// TIA Portal V18 export
DATA_BLOCK "Var_HMI"   // DB10
{ S7_Optimized_Access := 'FALSE' }
VERSION : 0.1
// stored: AutoNumber true, IsOnlyStoredInLoadMemory false, IsWriteProtectedInAS false
   VAR
      "popup Emergency" : Bool;
      "popup warning" : Bool;
      Selector : UInt := 5;
      "page number" : UInt := 12;
      in_selection : Bool;
      emergency_popup : Bool;
      selection_no : Int;
      scrolling_1 : Int;
      scrolling_2 : Int;
   END_VAR
BEGIN
END_DATA_BLOCK
